GLOBALCONSTANTS MessageExchangeConst (* All message values from the "Message exchange between services" sequence chart (Module 6, slides 42-46) *)
  (* Standard: 61499-1; Description: Copyright (c) 2026 Meisterschulen am Ostbahnhof This program and the accompanying materials are made available under the terms of the Eclipse Public License 2.0 which is available at https://www.eclipse.org/legal/epl-2.0/ SPDX-License-Identifier: EPL-2.0 *)
  (* Version 1.0, 2026-09-02, Franz Höpfinger, Meisterschulen am Ostbahnhof, Handshake design pattern (IEC 61499 primer course, Module 6, Valeriy Vyatkin), slides 42-46 "Message exchange between services" (five build/reveal states of the same diagram, content identical throughout) - every distinct REQ/RSP string value from the CylH/MES/WPS/DS message-sequence chart, extracted as named constants for the CylH message-exchange demo *)
  PACKAGE Meins::DesingPatterns::HandshakePattern::const;
  VAR_GLOBAL CONSTANT
    REQ_TRIP : WSTRING := "trip"; (* MES to CYL: perform the round trip *)
    REQ_EXTEND : WSTRING := "100"; (* CYL to CYL.push/CYL.pop: extend to 100 *)
    REQ_RETRACT : WSTRING := "0"; (* CYL to CYL.push/CYL.pop: retract to 0 *)
    REQ_DROP : WSTRING := "drop"; (* CYL to DS: drop the workpiece *)
    RSP_WPS_ABSENT : WSTRING := "WPS,0"; (* WPS: no workpiece present *)
    RSP_WPS_ARRIVED : WSTRING := "WPS,1"; (* WPS: workpiece arrived *)
    RSP_START_TRIGGERED : WSTRING := "start,1"; (* CYL.start: start-position sensor triggered *)
    RSP_END_IDLE : WSTRING := "end,0"; (* CYL.end: end-position sensor idle (not triggered) *)
    RSP_END_TRIGGERED : WSTRING := "end,1"; (* CYL.end: end-position sensor triggered *)
    RSP_PUSH_EXTENDED : WSTRING := "push,100"; (* CYL.push: push valve extended (100) *)
    RSP_PUSH_RETRACTED : WSTRING := "push,0"; (* CYL.push: push valve retracted (0) *)
    RSP_POP_EXTENDED : WSTRING := "pop,100"; (* CYL.pop: pop valve extended (100) *)
    RSP_POP_RETRACTED : WSTRING := "pop,0"; (* CYL.pop: pop valve retracted (0) *)
    RSP_CYL_STARTED : WSTRING := "CYL,STARTED"; (* CYL to MES: round trip started *)
    RSP_CYL_END_POS : WSTRING := "CYL, END POS"; (* CYL to MES: pusher reached end position *)
    RSP_CYL_START_POS : WSTRING := "CYL, START POS"; (* CYL to MES: pusher reached start position *)
    RSP_CYL_TRIP_COMPLETE : WSTRING := "CYL, Trip Complete"; (* CYL to MES: round trip service completed *)
    RSP_ACK : WSTRING := "ack"; (* DS to CYL: drop acknowledged *)
  END_VAR
END_GLOBALCONSTANTS
